Universal Robots PolyScope program: gravityFeederZ.urp

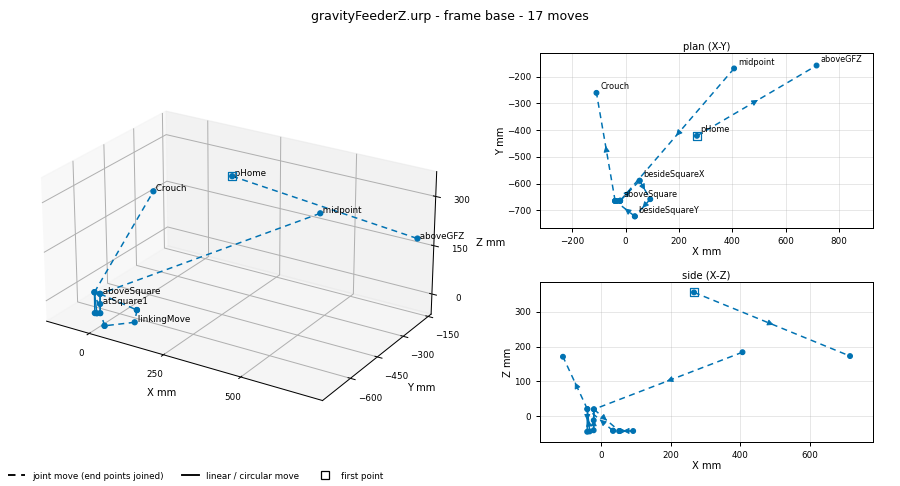
[picture p0: tool path of gravityFeederZ.urp in frame base, 17 of 22 moves have a stored position in this frame; points joined in program order, loops and branches not executed]
Program gravityFeederZ (installation=admin directory=/programs/WED_9AM createdIn=3.8.0.61336 lastSavedIn=3.15.8.106339 robotSerialNumber=2015350924)
Calibrated DH parameters: a=[0, -0.425, -0.39225, 0, 0, 0]; d=[0.089159, 0, 0, 0.10915, 0.09465, 0.0823]; alpha=[1.570796, 0, 0, 1.570796, -1.570796, 0]; deltaTheta=[0, 0, 0, 0, 0, 0]
Robot Program (runOnlyOnce=true)
  Set DigitalOutput pin=digital_out[0]; digitalValue=0
  Call _adminLinearIndex2
  MoveJ speed 180 deg/s, acceleration 100 deg/s^2 (useActiveTCP=true)
    Waypoint pHome: TCP in base x=267.118 y=-421.457 z=355.823 mm, rx=1.114 ry=1.1062 rz=0.0051 rad; joints [-44.998, -90.002, -90.001, -90.005, 90.001, 0.003] deg; flange x=267.125 y=-421.465 z=431.823 mm, rx=1.2022 ry=-2.9024 rz=-0.0002 rad
    Waypoint aboveGFZ: TCP in base x=715.199 y=-158.118 z=172.881 mm, rx=0.8748 ry=0.8572 rz=-0.013 rad; joints [-0.844, -122.124, -80.393, -53.429, 75.957, 43.451] deg; flange x=697.57 y=-139.415 z=244.403 mm, rx=-1.1146 ry=2.7612 rz=-0.4833 rad
  MoveL speed 150 mm/s, acceleration 50 mm/s^2 (useActiveTCP=true) feature=Base
    Waypoint atGFRel (Relative): relativeFromPosition TCP in base x=715.215 y=-158.048 z=172.914 mm, rx=0.8752 ry=0.8572 rz=-0.0126 rad; joints [-0.844, -122.122, -80.39, -53.429, 75.983, 43.452] deg; TCP in base x=733.158 y=-176.576 z=102.138 mm, rx=0.8753 ry=0.8572 rz=-0.0127 rad; joints [-2.339, -129.026, -80.24, -46.322, 76.352, 41.964] deg; flange x=715.523 y=-157.908 z=173.668 mm, rx=-1.1145 ry=2.7611 rz=-0.4826 rad
    Set DigitalOutput pin=digital_out[0]; digitalValue=1
    Wait Sleep waitTime=1
    Waypoint moveUpRel (Relative): relativeFromPosition TCP in base x=733.18 y=-176.563 z=102.148 mm, rx=0.8752 ry=0.8572 rz=-0.0127 rad; joints [-2.338, -129.027, -80.236, -46.322, 76.35, 41.964] deg; TCP in base x=735.26 y=-178.559 z=103.271 mm, rx=0.8752 ry=0.8572 rz=-0.0125 rad; joints [-2.494, -129.252, -79.66, -46.633, 76.392, 41.8] deg; flange x=717.617 y=-159.892 z=174.799 mm, rx=-1.1147 ry=2.7609 rz=-0.4827 rad
    Waypoint aboveGFRel (Relative): relativeFromPosition TCP in base x=735.253 y=-178.53 z=103.244 mm, rx=0.8752 ry=0.8573 rz=-0.0125 rad; joints [-2.492, -129.253, -79.661, -46.636, 76.392, 41.802] deg; TCP in base x=723.211 y=-166.183 z=150.627 mm, rx=0.8753 ry=0.8571 rz=-0.0126 rad; joints [-1.512, -124.544, -79.988, -51.245, 76.148, 42.788] deg; flange x=705.568 y=-147.516 z=222.156 mm, rx=-1.1145 ry=2.761 rz=-0.4826 rad
  MoveJ speed 180 deg/s, acceleration 100 deg/s^2 (useActiveTCP=true)
    Waypoint midpoint: TCP in base x=406.395 y=-169.035 z=183.96 mm, rx=1.0403 ry=1.0593 rz=0.0743 rad; joints [-7.736, -85.766, -121.496, -57.713, 88.681, 33.967] deg; flange x=400.037 y=-166.406 z=259.648 mm, rx=-1.2576 ry=2.8089 rz=-0.1014 rad
    Waypoint aboveSquare: TCP in base x=-20.27 y=-664.433 z=20.034 mm, rx=1.707 ry=-0.0117 rz=-1.2066 rad; joints [-82.307, -127.318, -92.1, -50.434, 90.041, 52.933] deg; flange x=-20.35 y=-664.245 z=96.034 mm, rx=1.2076 ry=2.8982 rz=-0.0029 rad
  MoveL speed 250 mm/s, acceleration 1200 mm/s^2 (useActiveTCP=true) feature=Base
    Waypoint atSquare1: TCP in base x=-20.834 y=-664.896 z=-11.616 mm, rx=1.7066 ry=-0.0121 rz=-1.2064 rad; joints [-82.362, -130.177, -92.819, -46.823, 90.046, 52.878] deg; flange x=-20.927 y=-664.667 z=64.384 mm, rx=1.2074 ry=2.8978 rz=-0.0036 rad
    Waypoint atSquare2: TCP in base x=-21.028 y=-665.074 z=-40.282 mm, rx=1.7065 ry=-0.0118 rz=-1.2061 rad; joints [-82.381, -132.91, -93.207, -43.701, 90.045, 52.836] deg; flange x=-21.119 y=-664.844 z=35.717 mm, rx=1.2068 ry=2.8981 rz=-0.0037 rad
    Set DigitalOutput pin=digital_out[0]; digitalValue=0
    Wait Sleep waitTime=0.5
    Waypoint aboveSquare: TCP in base x=-20.27 y=-664.433 z=20.034 mm, rx=1.707 ry=-0.0117 rz=-1.2066 rad; joints [-82.307, -127.318, -92.1, -50.434, 90.041, 52.933] deg; flange x=-20.35 y=-664.245 z=96.034 mm, rx=1.2076 ry=2.8982 rz=-0.0029 rad
    Set DigitalOutput pin=digital_out[0]; digitalValue=1
  MoveJ speed 60 deg/s, acceleration 80 deg/s^2 (useActiveTCP=true)
    Waypoint besideSquareX: TCP in base x=52.617 y=-589.571 z=-42.423 mm, rx=1.7065 ry=-0.0117 rz=-1.2076 rad; joints [-74.267, -126.531, -106.897, -36.426, 89.974, 61.001] deg; flange x=52.598 y=-589.375 z=33.577 mm, rx=1.2085 ry=2.8985 rz=-0.0036 rad
  MoveL speed 35 mm/s, acceleration 35 mm/s^2 (useActiveTCP=true) feature=Base
    If force()≤40 (checkContinuously=true)
      Waypoint atSquareX (Relative): relativeFromPosition TCP in base x=50.865 y=-591.008 z=-41.515 mm, rx=1.7022 ry=-0.008 rz=-1.2089 rad; joints [-74.266, -126.532, -106.898, -36.426, 89.971, 60.977] deg; TCP in base x=-28.314 y=-672.475 z=-41.562 mm, rx=1.7067 ry=-0.0121 rz=-1.2064 rad; joints [-83.089, -133.766, -91.707, -44.351, 90.046, 52.151] deg; flange x=-28.404 y=-672.249 z=34.438 mm, rx=1.2075 ry=2.8979 rz=-0.0036 rad
    Wait Sleep waitTime=0.5
  MoveJ speed 60 deg/s, acceleration 80 deg/s^2 (useActiveTCP=true)
    Waypoint besideSquareX: TCP in base x=52.617 y=-589.571 z=-42.423 mm, rx=1.7065 ry=-0.0117 rz=-1.2076 rad; joints [-74.267, -126.531, -106.897, -36.426, 89.974, 61.001] deg; flange x=52.598 y=-589.375 z=33.577 mm, rx=1.2085 ry=2.8985 rz=-0.0036 rad
    Waypoint linkingMove: motionParameters(blendRadius=0.01); TCP in base x=92.406 y=-658.703 z=-42.29 mm, rx=1.7071 ry=-0.0114 rz=-1.2067 rad; joints [-72.572, -133.085, -93.255, -43.522, 90.01, 62.663] deg; flange x=92.339 y=-658.532 z=33.709 mm, rx=1.2075 ry=2.8984 rz=-0.0027 rad
    Waypoint besideSquareY: TCP in base x=34.628 y=-723.042 z=-41.53 mm, rx=1.7068 ry=-0.0118 rz=-1.2057 rad; joints [-78.597, -138.866, -81.159, -49.796, 90.051, 56.613] deg; flange x=34.515 y=-722.822 z=34.47 mm, rx=1.2066 ry=2.8979 rz=-0.0033 rad
  MoveL speed 35 mm/s, acceleration 35 mm/s^2 (useActiveTCP=true) feature=Base
    If force()≤40 (checkContinuously=true)
      Waypoint atSquareY (Relative): relativeFromPosition TCP in base x=32.384 y=-724.404 z=-40.504 mm, rx=1.7021 ry=-0.0085 rz=-1.209 rad; joints [-78.599, -138.865, -81.161, -49.795, 90.053, 56.612] deg; TCP in base x=-15.815 y=-673.74 z=-41.486 mm, rx=1.7062 ry=-0.0122 rz=-1.2065 rad; joints [-82.031, -133.838, -91.548, -44.418, 90.028, 53.212] deg; flange x=-15.889 y=-673.488 z=34.513 mm, rx=1.2075 ry=2.8979 rz=-0.0042 rad
    Wait Sleep waitTime=0.5
  MoveJ speed 60 deg/s, acceleration 80 deg/s^2 (useActiveTCP=true)
    Waypoint besideSquareY: TCP in base x=34.628 y=-723.042 z=-41.53 mm, rx=1.7068 ry=-0.0118 rz=-1.2057 rad; joints [-78.597, -138.866, -81.159, -49.796, 90.051, 56.613] deg; flange x=34.515 y=-722.822 z=34.47 mm, rx=1.2066 ry=2.8979 rz=-0.0033 rad
    Waypoint aboveSquareNew: TCP in base x=-39.171 y=-665.188 z=20.711 mm, rx=1.7064 ry=-0.0121 rz=-1.2063 rad; joints [-83.953, -127.424, -91.788, -50.601, 90.045, 51.279] deg; flange x=-39.256 y=-664.947 z=96.711 mm, rx=1.2072 ry=2.8979 rz=-0.0039 rad
    Set DigitalOutput pin=digital_out[0]; digitalValue=0
    Wait Sleep waitTime=1
  MoveL speed 250 mm/s, acceleration 1200 mm/s^2 (useActiveTCP=true) feature=Base
    Waypoint atSquareNew: TCP in base x=-39.623 y=-665.674 z=-44.47 mm, rx=1.7064 ry=-0.0122 rz=-1.2064 rad; joints [-83.996, -133.455, -92.966, -43.391, 90.044, 51.246] deg; flange x=-39.706 y=-665.432 z=31.529 mm, rx=1.2075 ry=2.8978 rz=-0.004 rad
    Set DigitalOutput pin=digital_out[0]; digitalValue=1
    Wait Sleep waitTime=1
    Waypoint easeout: TCP in base x=-32.563 y=-665.585 z=-43.483 mm, rx=1.7065 ry=-0.0122 rz=-1.2064 rad; joints [-83.384, -133.314, -93.049, -43.45, 90.044, 51.855] deg; flange x=-32.65 y=-665.346 z=32.516 mm, rx=1.2074 ry=2.8978 rz=-0.0039 rad
    Waypoint aboveSquareNew: TCP in base x=-39.171 y=-665.188 z=20.711 mm, rx=1.7064 ry=-0.0121 rz=-1.2063 rad; joints [-83.953, -127.424, -91.788, -50.601, 90.045, 51.279] deg; flange x=-39.256 y=-664.947 z=96.711 mm, rx=1.2072 ry=2.8979 rz=-0.0039 rad
  Call _adminLinearIndex4
  MoveJ speed 60 deg/s, acceleration 80 deg/s^2 (useActiveTCP=true)
    Waypoint Crouch: TCP in base x=-109.165 y=-260.498 z=170.953 mm, rx=1.6765 ry=0.1344 rz=-1.0824 rad; joints [-90.004, -61.53, -138.325, -70.319, 90.001, 35.527] deg; flange x=-109.166 y=-260.729 z=246.952 mm, rx=-0.9583 ry=-2.9909 rz=-0.0046 rad
SubProgram -> _adminLinearIndex4
SubProgram  [hidden by the author, left out]
SubProgram _adminLinearIndex2 [hidden by the author, left out]
SubProgram _adminLinearIndex4 (keepSynchronizedWithDisk=false) programFile=/programs/me345_admin/_adminLinearIndex4.urp
  Folder Move_linear_slide_Index4
    var_1 := False
    Loop While (checkContinuously=false) expression=var_1≟ False
      var_1 := socket_open("10.241.34.52",4001)
    var_3 := 1
    Send := "s r0x24 21"
    Script: socket_send_string(Send)
    Script: socket_send_byte(13)
    Send_Reply := socket_read_string()
    Send := "s r0xca 169167"
    Script: socket_send_string(Send)
    Script: socket_send_byte(13)
    Send_Reply := socket_read_string()
    Send := "t 1"
    Script: socket_send_string(Send)
    Script: socket_send_byte(13)
    Send_Reply := socket_read_string()
    Loop While (checkContinuously=false) expression=var_3≠0
      Send := "g r0xA0"
      Script: socket_send_string(Send)
      Script: socket_send_byte(13)
      var_3 := socket_get_var("v")
      Wait Sleep waitTime=0.1
    Script: socket_close()
    Script: sync()
